{attribute 'strict'}
TYPE E_GoldenSampleState :
(
	GS_STATUS_UNKNOWN		:= 0,
	GS_STATUS_BCHECKSETUP	:= 10,
	GS_STATUS_NOK			:= 20,
	GS_STATUS_OK			:= 30
);
END_TYPE

(* stored: Version 1.1.0.1, ProductVersion 3.1.4024.9
   DUT E_GoldenSampleState: Id {17d267d4-00e2-4f4e-8c62-927dcfa2f118} *)
